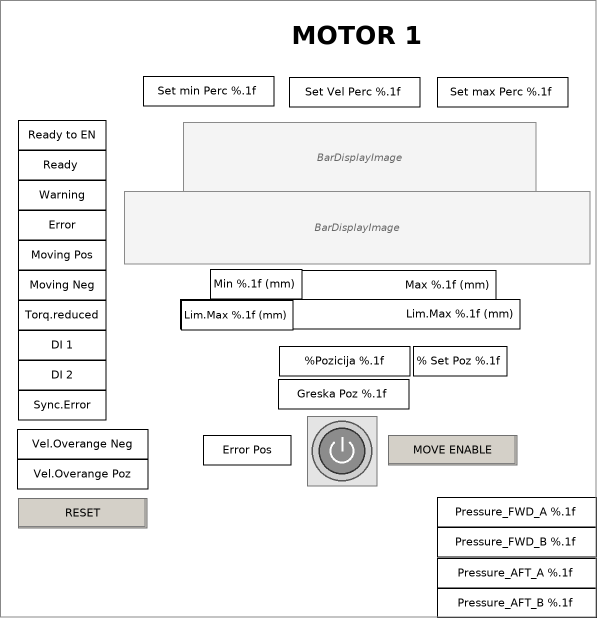
VISUALIZATION VisuDoorControl  // 597x618
    Rectangle (210,270 286x30), "Max %.1f (mm)", text variable: MAIN.FB_DC_MOTOR1.rRadno_Max_Pos
        OnMouseDown: write the text variable via Default, min 0, max 100
    PowerSwitch (307,416 70x70), variable: PRG_ZF_Control.bMotorOn_M1, behaviour: TOGGLE, style: Switch-PowerSwitch-Gray
    Rectangle (143,76 131x30), "Set min Perc %.1f", text variable: MAIN.rSetpointTarget_MinM1
        OnMouseDown: write the text variable via Default, min 0, max 100
    Rectangle (437,77 131x30), "Set max Perc %.1f", text variable: MAIN.rSetpointTarget_MaxM1
        OnMouseDown: write the text variable via Default, min 0, max 100
    Rectangle (279,346 131x30), "%Pozicija %.1f", text variable: MAIN.rPotFeedback_Radno_PercM1
    Rectangle (289,77 131x30), "Set Vel Perc %.1f", text variable: MAIN.rMaxVelocityM1
        OnMouseDown: write the text variable via Default, min 0, max 120
    Rectangle (278,379 131x30), "Greska Poz %.1f", text variable: MAIN.rErrorM1, colour toggle: MAIN.bInDeadband_M1
    Rectangle (413,346 94x30), "% Set Poz %.1f", text variable: MAIN.rSetpointTarget_M1
        OnMouseDown: write the text variable via Default, min 0, max 100
    Rectangle (17,429 131x30), "Vel.Overange Neg", colour toggle: MAIN.FB_DC_MOTOR1.bSetVelOverNeg
    Rectangle (17,459 131x30), "Vel.Overange Poz", colour toggle: MAIN.FB_DC_MOTOR1.bSetVelOverPoz
    Button (18,498 129x30), "RESET"
        tap MAIN.bHMI_RESET_M1
    Rectangle (18,120 88x30), "Ready to EN", colour toggle: bReadyToEnable_M1
    Rectangle (18,150 88x30), "Ready", colour toggle: bReady_M1
    Rectangle (18,180 88x30), "Warning", colour toggle: bWarning_M1
    Rectangle (18,210 88x30), "Error", colour toggle: bError_M1
    Rectangle (18,240 88x30), "Moving Pos", colour toggle: bMovingPositive_M1
    Rectangle (18,270 88x30), "Moving Neg", colour toggle: bMovingNegative_M1
    Rectangle (18,300 88x30), "Torq.reduced", colour toggle: bTorqueReduced_M1
    Rectangle (18,330 88x30), "DI 1", colour toggle: bDigitalInput1_M1
    Rectangle (18,360 88x30), "DI 2", colour toggle: bDigitalInput2_M1
    Rectangle (18,390 88x30), "Sync.Error", colour toggle: bSyncError_M1
    Button (388,435 129x30), "MOVE ENABLE", colour toggle: MAIN.bMove_M1
        toggle MAIN.bMove_M1
    BarDisplayImage (183,122 353x71), value: PRG_ZF_Control.rPotFeedback_Radno_PercM1, style: BarDisplayImage-Gray, scale format: %.1f, scale 0..100
        p518627256: %
    BarDisplayImage (124,191 466x73), value: PRG_ZF_Control.FB_DC_MOTOR1.rLinearPosition, style: BarDisplayImage-Gray, scale format: %.1f, scale 0..80
        p518627256: mm
    Rectangle (210,269 92x30), "Min %.1f (mm)", text variable: MAIN.FB_DC_MOTOR1.rRadno_Min_Pos
        OnMouseDown: write the text variable via Default, min 0, max 100
    Rectangle (180,299 340x30), "Lim.Max %.1f (mm)", text variable: MAIN.FB_DC_MOTOR1.rLinearPosition_LimMAx, colour toggle: MAIN.bErrorLimitPosMax_M1
        OnMouseDown: write the text variable via Default, min 0, max 100
    Rectangle (181,300 112x30), "Lim.Max %.1f (mm)", text variable: MAIN.FB_DC_MOTOR1.rLinearPosition_LimMin, colour toggle: MAIN.bErrorLimitPosMin_M1
        OnMouseDown: write the text variable via Default, min 0, max 100
    Label (146,20 422x30), "MOTOR 1"
    Rectangle (203,435 88x30), "Error Pos", colour toggle: MAIN.bERROR_POS_M1
    Rectangle (437,497 160x30), "Pressure_FWD_A %.1f", text variable: GVL_IO.fPressure_FWD_A
    Rectangle (437,527 160x30), "Pressure_FWD_B %.1f", text variable: GVL_IO.fPressure_FWD_B
    Rectangle (437,558 160x30), "Pressure_AFT_A %.1f", text variable: GVL_IO.fPressure_AFT_A
    Rectangle (437,588 160x30), "Pressure_AFT_B %.1f", text variable: GVL_IO.fPressure_AFT_B
END_VISUALIZATION

(* stored: Version 1.1.0.1, ProductVersion 3.1.4026.17
   Visu VisuDoorControl: Id {4e47eb22-7868-425b-91e5-15251edd3ae0} *)
